(* Logix 5000 project; controller Final vendor 1 type 14 code 242 rev 32.11; software revision 32.00 *)

TASK InitializationTask (periodic, rate 10 ms, priority 10, watchdog 500 ms) : InitializationProgram   // Initializes the tags with default values
TASK MainTask (continuous, watchdog 500 ms) : MainProgram
TASK ProcessDataTask (periodic, rate 10 ms, priority 10, watchdog 500 ms) : ProcessDataI   // Processes the data that has been read and determines the next steps of the pod
TASK ReadTask (periodic, rate 10 ms, priority 10, watchdog 500 ms) : UpdatePrev, UpdateCurrent   // Task that reads current sensor values without erasing previous sensor values
TASK SafetyTask (periodic, rate 20 ms, priority 10, watchdog 20 ms, safety) : SafetyProgram

MODULES
   Local : vendor 1 type 14 code 242 (5069 0, rev 32.11)
      IO_002 : 5069-IF8 (5069 2, rev 2.1, StandardDataDriven RPI 100 ms)
      IO_001 : 5069-IF8 (5069 1, rev 2.1, StandardDataDriven RPI 100 ms)
      IO_003 : 5069-IF8 (5069 3, rev 2.1, StandardDataDriven RPI 100 ms)
      IO_006 : vendor 1 type 7 code 394 (5069 6, rev 2.1, StandardDataDriven RPI 5 ms)
      IO_004 : vendor 1 type 7 code 395 (5069 4, rev 2.1, StandardDataDriven RPI 5 ms)
      IO_005 : vendor 1 type 7 code 395 (5069 5, rev 2.1, StandardDataDriven RPI 5 ms)
      IO_007 : vendor 1 type 109 code 90 (5069 7, rev 3.1, StandardDataDriven RPI 80 ms)
      EN_001 : 1734-AENTR (Ethernet 107.0.114.14, rev 5.1, Output RPI 20 ms)
END_MODULES

TYPE SensorType :   // To monitor the sensor readings, we use this data type
STRUCT
   CurrentValue : DINT;
   PreviousValue0 : DINT;
   PreviousValue1 : DINT;
   PreviousValue2 : DINT;
   PreviousValue3 : DINT;
   PreviousValue4 : DINT;
   PreviousValue5 : DINT;
   PreviousValue6 : DINT;
   PreviousValue7 : DINT;
   PreviousValue8 : DINT;
   PreviousValue9 : DINT;
   Mean10 : DINT;
   StanDev : DINT;
   State : DINT;
   Count : DINT;
END_STRUCT
END_TYPE

VAR_GLOBAL   (* controller tags *)
   B_Pres0 : SensorType;   // Holds all values related to Brakes Pressure Sensor #0
   B_Pres1 : SensorType;   // Holds all values related to Brakes Pressure Sensor #1
   B_Pres2 : SensorType;   // Holds all values related to Brakes Pressure Sensor #2
   B_Pres3 : SensorType;   // Holds all values related to Brakes Pressure Sensor #3
   B_Pres4 : SensorType;   // Holds all values related to Brakes Pressure Sensor #4
   B_Pres5 : SensorType;   // Holds all values related to Brakes Pressure Sensor #5
   B_Pres6 : SensorType;   // Holds all values related to Brakes Pressure Sensor #6
   B_Pres7 : SensorType;   // Holds all values related to Brakes Pressure Sensor #7
   B_Pres8 : SensorType;   // Holds all values related to Brakes Pressure Sensor #8
   B_Pres9 : SensorType;   // Holds all values related to Brakes Pressure Sensor #9
   B_Tem0 : SensorType;   // Holds all values related to Brakes Temperature Sensor #0
   B_Tem1 : SensorType;   // Holds all values related to Brakes Temperature Sensor #1
   C_Las0 : SensorType;   // Holds all values related to Controls Laser Sensor #0
   C_Las1 : SensorType;   // Holds all values related to Controls Laser Sensor #1
   CurrentState : DINT;
   P_Pres0 : SensorType;   // Holds all values related to Pressure Pressure Sensor #0
   P_Pres1 : SensorType;   // Holds all values related to Pressure Pressure Sensor #1
   P_Pres2 : SensorType;   // Holds all values related to Pressure Pressure Sensor #2
   P_Tem0 : SensorType;   // Holds all values related to Pressure Temperature Sensor #0
   P_Tem1 : SensorType;   // Holds all values related to Pressure Temperature Sensor #1
END_VAR

PROGRAM InitializationProgram   (* main routine Initial_B_Pres0 *)

ROUTINE Initial_B_Pres0   (* structured text *)
   B_Pres0.CurrentValue := 0;
   B_Pres0.PreviousValue0 := 0;
   B_Pres0.PreviousValue1 := 0;
   B_Pres0.PreviousValue2 := 0;
   B_Pres0.PreviousValue3 := 0;
   B_Pres0.PreviousValue4 := 0;
   B_Pres0.PreviousValue5 := 0;
   B_Pres0.PreviousValue6 := 0;
   B_Pres0.PreviousValue7 := 0;
   B_Pres0.PreviousValue8 := 0;
   B_Pres0.PreviousValue9 := 0;
   B_Pres0.Count := 0;
   B_Pres0.Mean10 := 0;
   B_Pres0.StanDev := 0;
   B_Pres0.State := 0;
END_ROUTINE

ROUTINE Initial_B_Pres1   (* structured text *)
   B_Pres1.CurrentValue := 0;
   B_Pres1.PreviousValue0 := 0;
   B_Pres1.PreviousValue1 := 0;
   B_Pres1.PreviousValue2 := 0;
   B_Pres1.PreviousValue3 := 0;
   B_Pres1.PreviousValue4 := 0;
   B_Pres1.PreviousValue5 := 0;
   B_Pres1.PreviousValue6 := 0;
   B_Pres1.PreviousValue7 := 0;
   B_Pres1.PreviousValue8 := 0;
   B_Pres1.PreviousValue9 := 0;
   B_Pres1.Count := 0;
   B_Pres1.Mean10 := 0;
   B_Pres1.StanDev := 0;
   B_Pres1.State := 0;
END_ROUTINE

ROUTINE Initial_B_Pres2   (* structured text *)
   B_Pres2.CurrentValue := 0;
   B_Pres2.PreviousValue0 := 0;
   B_Pres2.PreviousValue1 := 0;
   B_Pres2.PreviousValue2 := 0;
   B_Pres2.PreviousValue3 := 0;
   B_Pres2.PreviousValue4 := 0;
   B_Pres2.PreviousValue5 := 0;
   B_Pres2.PreviousValue6 := 0;
   B_Pres2.PreviousValue7 := 0;
   B_Pres2.PreviousValue8 := 0;
   B_Pres2.PreviousValue9 := 0;
   B_Pres2.Count := 0;
   B_Pres2.Mean10 := 0;
   B_Pres2.StanDev := 0;
   B_Pres2.State := 0;
END_ROUTINE

ROUTINE Initial_B_Pres3   (* structured text *)
   B_Pres3.CurrentValue := 0;
   B_Pres3.PreviousValue0 := 0;
   B_Pres3.PreviousValue1 := 0;
   B_Pres3.PreviousValue2 := 0;
   B_Pres3.PreviousValue3 := 0;
   B_Pres3.PreviousValue4 := 0;
   B_Pres3.PreviousValue5 := 0;
   B_Pres3.PreviousValue6 := 0;
   B_Pres3.PreviousValue7 := 0;
   B_Pres3.PreviousValue8 := 0;
   B_Pres3.PreviousValue9 := 0;
   B_Pres3.Count := 0;
   B_Pres3.Mean10 := 0;
   B_Pres3.StanDev := 0;
   B_Pres3.State := 0;
END_ROUTINE

ROUTINE Initial_B_Pres4   (* structured text *)
   B_Pres4.CurrentValue := 0;
   B_Pres4.PreviousValue0 := 0;
   B_Pres4.PreviousValue1 := 0;
   B_Pres4.PreviousValue2 := 0;
   B_Pres4.PreviousValue3 := 0;
   B_Pres4.PreviousValue4 := 0;
   B_Pres4.PreviousValue5 := 0;
   B_Pres4.PreviousValue6 := 0;
   B_Pres4.PreviousValue7 := 0;
   B_Pres4.PreviousValue8 := 0;
   B_Pres4.PreviousValue9 := 0;
   B_Pres4.Count := 0;
   B_Pres4.Mean10 := 0;
   B_Pres4.StanDev := 0;
   B_Pres4.State := 0;
END_ROUTINE

ROUTINE Initial_B_Pres5   (* structured text *)
   B_Pres5.CurrentValue := 0;
   B_Pres5.PreviousValue0 := 0;
   B_Pres5.PreviousValue1 := 0;
   B_Pres5.PreviousValue2 := 0;
   B_Pres5.PreviousValue3 := 0;
   B_Pres5.PreviousValue4 := 0;
   B_Pres5.PreviousValue5 := 0;
   B_Pres5.PreviousValue6 := 0;
   B_Pres5.PreviousValue7 := 0;
   B_Pres5.PreviousValue8 := 0;
   B_Pres5.PreviousValue9 := 0;
   B_Pres5.Count := 0;
   B_Pres5.Mean10 := 0;
   B_Pres5.StanDev := 0;
   B_Pres5.State := 0;
END_ROUTINE

ROUTINE Initial_B_Pres6   (* structured text *)
   B_Pres6.CurrentValue := 0;
   B_Pres6.PreviousValue0 := 0;
   B_Pres6.PreviousValue1 := 0;
   B_Pres6.PreviousValue2 := 0;
   B_Pres6.PreviousValue3 := 0;
   B_Pres6.PreviousValue4 := 0;
   B_Pres6.PreviousValue5 := 0;
   B_Pres6.PreviousValue6 := 0;
   B_Pres6.PreviousValue7 := 0;
   B_Pres6.PreviousValue8 := 0;
   B_Pres6.PreviousValue9 := 0;
   B_Pres6.Count := 0;
   B_Pres6.Mean10 := 0;
   B_Pres6.StanDev := 0;
   B_Pres6.State := 0;
END_ROUTINE

ROUTINE Initial_B_Pres7   (* structured text *)
   B_Pres7.CurrentValue := 0;
   B_Pres7.PreviousValue0 := 0;
   B_Pres7.PreviousValue1 := 0;
   B_Pres7.PreviousValue2 := 0;
   B_Pres7.PreviousValue3 := 0;
   B_Pres7.PreviousValue4 := 0;
   B_Pres7.PreviousValue5 := 0;
   B_Pres7.PreviousValue6 := 0;
   B_Pres7.PreviousValue7 := 0;
   B_Pres7.PreviousValue8 := 0;
   B_Pres7.PreviousValue9 := 0;
   B_Pres7.Count := 0;
   B_Pres7.Mean10 := 0;
   B_Pres7.StanDev := 0;
   B_Pres7.State := 0;
END_ROUTINE

ROUTINE Initial_B_Pres8   (* structured text *)
   B_Pres8.CurrentValue := 0;
   B_Pres8.PreviousValue0 := 0;
   B_Pres8.PreviousValue1 := 0;
   B_Pres8.PreviousValue2 := 0;
   B_Pres8.PreviousValue3 := 0;
   B_Pres8.PreviousValue4 := 0;
   B_Pres8.PreviousValue5 := 0;
   B_Pres8.PreviousValue6 := 0;
   B_Pres8.PreviousValue7 := 0;
   B_Pres8.PreviousValue8 := 0;
   B_Pres8.PreviousValue9 := 0;
   B_Pres8.Count := 0;
   B_Pres8.Mean10 := 0;
   B_Pres8.StanDev := 0;
   B_Pres8.State := 0;
END_ROUTINE

ROUTINE Initial_B_Pres9   (* structured text *)
   B_Pres9.CurrentValue := 0;
   B_Pres9.PreviousValue0 := 0;
   B_Pres9.PreviousValue1 := 0;
   B_Pres9.PreviousValue2 := 0;
   B_Pres9.PreviousValue3 := 0;
   B_Pres9.PreviousValue4 := 0;
   B_Pres9.PreviousValue5 := 0;
   B_Pres9.PreviousValue6 := 0;
   B_Pres9.PreviousValue7 := 0;
   B_Pres9.PreviousValue8 := 0;
   B_Pres9.PreviousValue9 := 0;
   B_Pres9.Count := 0;
   B_Pres9.Mean10 := 0;
   B_Pres9.StanDev := 0;
   B_Pres9.State := 0;
END_ROUTINE

ROUTINE Initial_B_Tem0   (* structured text *)
   B_Tem0.CurrentValue := 0;
   B_Tem0.PreviousValue0 := 0;
   B_Tem0.PreviousValue1 := 0;
   B_Tem0.PreviousValue2 := 0;
   B_Tem0.PreviousValue3 := 0;
   B_Tem0.PreviousValue4 := 0;
   B_Tem0.PreviousValue5 := 0;
   B_Tem0.PreviousValue6 := 0;
   B_Tem0.PreviousValue7 := 0;
   B_Tem0.PreviousValue8 := 0;
   B_Tem0.PreviousValue9 := 0;
   B_Tem0.Count := 0;
   B_Tem0.Mean10 := 0;
   B_Tem0.StanDev := 0;
   B_Tem0.State := 0;
END_ROUTINE

ROUTINE Initial_B_Tem1   (* structured text *)
   B_Tem1.CurrentValue := 0;
   B_Tem1.PreviousValue0 := 0;
   B_Tem1.PreviousValue1 := 0;
   B_Tem1.PreviousValue2 := 0;
   B_Tem1.PreviousValue3 := 0;
   B_Tem1.PreviousValue4 := 0;
   B_Tem1.PreviousValue5 := 0;
   B_Tem1.PreviousValue6 := 0;
   B_Tem1.PreviousValue7 := 0;
   B_Tem1.PreviousValue8 := 0;
   B_Tem1.PreviousValue9 := 0;
   B_Tem1.Count := 0;
   B_Tem1.Mean10 := 0;
   B_Tem1.StanDev := 0;
   B_Tem1.State := 0;
END_ROUTINE

ROUTINE Initial_C_Las0   (* structured text *)
   C_Las0.CurrentValue := 0;
   C_Las0.PreviousValue0 := 0;
   C_Las0.PreviousValue1 := 0;
   C_Las0.PreviousValue2 := 0;
   C_Las0.PreviousValue3 := 0;
   C_Las0.PreviousValue4 := 0;
   C_Las0.PreviousValue5 := 0;
   C_Las0.PreviousValue6 := 0;
   C_Las0.PreviousValue7 := 0;
   C_Las0.PreviousValue8 := 0;
   C_Las0.PreviousValue9 := 0;
   C_Las0.Count := 0;
   C_Las0.Mean10 := 0;
   C_Las0.StanDev := 0;
   C_Las0.State := 0;
END_ROUTINE

ROUTINE Initial_C_Las1   (* structured text *)
   C_Las1.CurrentValue := 0;
   C_Las1.PreviousValue0 := 0;
   C_Las1.PreviousValue1 := 0;
   C_Las1.PreviousValue2 := 0;
   C_Las1.PreviousValue3 := 0;
   C_Las1.PreviousValue4 := 0;
   C_Las1.PreviousValue5 := 0;
   C_Las1.PreviousValue6 := 0;
   C_Las1.PreviousValue7 := 0;
   C_Las1.PreviousValue8 := 0;
   C_Las1.PreviousValue9 := 0;
   C_Las1.Count := 0;
   C_Las1.Mean10 := 0;
   C_Las1.StanDev := 0;
   C_Las1.State := 0;
END_ROUTINE

ROUTINE Initial_P_Pres0   (* structured text *)
   P_Pres0.CurrentValue := 0;
   P_Pres0.PreviousValue0 := 0;
   P_Pres0.PreviousValue1 := 0;
   P_Pres0.PreviousValue2 := 0;
   P_Pres0.PreviousValue3 := 0;
   P_Pres0.PreviousValue4 := 0;
   P_Pres0.PreviousValue5 := 0;
   P_Pres0.PreviousValue6 := 0;
   P_Pres0.PreviousValue7 := 0;
   P_Pres0.PreviousValue8 := 0;
   P_Pres0.PreviousValue9 := 0;
   P_Pres0.Count := 0;
   P_Pres0.Mean10 := 0;
   P_Pres0.StanDev := 0;
   P_Pres0.State := 0;
END_ROUTINE

ROUTINE Initial_P_Pres1   (* structured text *)
   P_Pres1.CurrentValue := 0;
   P_Pres1.PreviousValue0 := 0;
   P_Pres1.PreviousValue1 := 0;
   P_Pres1.PreviousValue2 := 0;
   P_Pres1.PreviousValue3 := 0;
   P_Pres1.PreviousValue4 := 0;
   P_Pres1.PreviousValue5 := 0;
   P_Pres1.PreviousValue6 := 0;
   P_Pres1.PreviousValue7 := 0;
   P_Pres1.PreviousValue8 := 0;
   P_Pres1.PreviousValue9 := 0;
   P_Pres1.Count := 0;
   P_Pres1.Mean10 := 0;
   P_Pres1.StanDev := 0;
   P_Pres1.State := 0;
END_ROUTINE

ROUTINE Initial_P_Pres2   (* structured text *)
   P_Pres2.CurrentValue := 0;
   P_Pres2.PreviousValue0 := 0;
   P_Pres2.PreviousValue1 := 0;
   P_Pres2.PreviousValue2 := 0;
   P_Pres2.PreviousValue3 := 0;
   P_Pres2.PreviousValue4 := 0;
   P_Pres2.PreviousValue5 := 0;
   P_Pres2.PreviousValue6 := 0;
   P_Pres2.PreviousValue7 := 0;
   P_Pres2.PreviousValue8 := 0;
   P_Pres2.PreviousValue9 := 0;
   P_Pres2.Count := 0;
   P_Pres2.Mean10 := 0;
   P_Pres2.StanDev := 0;
   P_Pres2.State := 0;
END_ROUTINE

ROUTINE Initial_P_Tem0   (* structured text *)
   P_Tem0.CurrentValue := 0;
   P_Tem0.PreviousValue0 := 0;
   P_Tem0.PreviousValue1 := 0;
   P_Tem0.PreviousValue2 := 0;
   P_Tem0.PreviousValue3 := 0;
   P_Tem0.PreviousValue4 := 0;
   P_Tem0.PreviousValue5 := 0;
   P_Tem0.PreviousValue6 := 0;
   P_Tem0.PreviousValue7 := 0;
   P_Tem0.PreviousValue8 := 0;
   P_Tem0.PreviousValue9 := 0;
   P_Tem0.Count := 0;
   P_Tem0.Mean10 := 0;
   P_Tem0.StanDev := 0;
   P_Tem0.State := 0;
END_ROUTINE

ROUTINE Initial_P_Tem1   (* structured text *)
   P_Tem1.CurrentValue := 0;
   P_Tem1.PreviousValue0 := 0;
   P_Tem1.PreviousValue1 := 0;
   P_Tem1.PreviousValue2 := 0;
   P_Tem1.PreviousValue3 := 0;
   P_Tem1.PreviousValue4 := 0;
   P_Tem1.PreviousValue5 := 0;
   P_Tem1.PreviousValue6 := 0;
   P_Tem1.PreviousValue7 := 0;
   P_Tem1.PreviousValue8 := 0;
   P_Tem1.PreviousValue9 := 0;
   P_Tem1.Count := 0;
   P_Tem1.Mean10 := 0;
   P_Tem1.StanDev := 0;
   P_Tem1.State := 0;
END_ROUTINE
END_PROGRAM

PROGRAM MainProgram   (* main routine MainRoutine *)

ROUTINE MainRoutine   (* ladder *)
END_ROUTINE
END_PROGRAM

PROGRAM ProcessDataI   (* main routine R001 *)
// Part-I of Process Data
VAR
   acceleration : DINT;
   crawl_distance_brake : DINT;
   distance : DINT;
   distance_brake : DINT;
   getDistance : DINT;
   nominal_count : DINT;
   prev_distance : DINT;
   prev_time : DINT;
   prev_velocity : DINT;
   temp_distance : DINT;
   time : DINT;
   velocity : DINT;
END_VAR

ROUTINE R001   (* structured text *)
   prev_time := time;
   prev_distance := distance;
   prev_velocity := velocity;
   time :=  TT;
   
   temp_distance := 0;
   nominal_count := 0;
   IF C_Las0.State = 0 THEN
               temp_distance :=  C_Las0.CurrentValue;
               nominal_count := 1;
   END_IF;
    IF C_Las1.State = 0 THEN
               temp_distance := temp_distance + C_Las1.CurrentValue;
               nominal_count := nominal_count + 1;
    END_IF;
   temp_distance := temp_distance / nominal_count;
   getDistance := temp_distance;
   
   distance := getDistance;
   velocity := (distance - prev_distance)/(time - prev_time);
   acceleration := (velocity - prev_velocity)/(time - prev_time);
END_ROUTINE

ROUTINE R002   (* structured text *)
   CASE EN_001:I.Data of
               1:  CurrentState := 1;
               2:  CurrentState := 0;
               3:  CurrentState := 2;
               4:  CurrentState := 3;
               6:  CurrentState := 5;
               8:  CurrentState := 6;
               10: CurrentState := 8;
    END_CASE;
END_ROUTINE

ROUTINE R003   (* structured text *)
   IF distance = (distance_brake) THEN
   	CurrentState := 5;
   ELSIF distance = (crawl_distance_brake) THEN
   	CurrentState := 5;
   //elsif timer
   END_IF;
    IF acceleration = 0 THEN
   	CurrentState := 4;
   //elsif timer
   END_IF;
   IF velocity = 0 THEN
   	CurrentState := 7;
   END_IF;
END_ROUTINE
END_PROGRAM

PROGRAM SafetyProgram   (* main routine MainRoutine, safety *)

ROUTINE MainRoutine   (* ladder *)
END_ROUTINE
END_PROGRAM

PROGRAM UpdateCurrent   (* main routine UC_B_Pres0 *)
// Program to store current sensor values
VAR
   range0 : DINT;
   range1 : DINT;
   range2 : DINT;
   range3 : DINT;
   range4 : DINT;
   range5 : DINT;
   range6 : DINT;
   range7 : DINT;
END_VAR

ROUTINE UC_B_Pres0   (* structured text *)
   B_Pres0.CurrentValue := Local:1:I.Ch00.Data;
END_ROUTINE

ROUTINE UC_B_Pres1   (* structured text *)
   B_Pres1.CurrentValue := Local:1:I.Ch01.Data;
END_ROUTINE

ROUTINE UC_B_Pres2   (* structured text *)
   B_Pres2.CurrentValue := Local:1:I.Ch02.Data;
END_ROUTINE

ROUTINE UC_B_Pres3   (* structured text *)
   B_Pres3.CurrentValue := Local:1:I.Ch03.Data;
END_ROUTINE

ROUTINE UC_B_Pres4   (* structured text *)
   B_Pres4.CurrentValue := Local:1:I.Ch04.Data;
END_ROUTINE

ROUTINE UC_B_Pres5   (* structured text *)
   B_Pres5.CurrentValue := Local:1:I.Ch05.Data;
END_ROUTINE

ROUTINE UC_B_Pres6   (* structured text *)
   B_Pres6.CurrentValue := Local:1:I.Ch06.Data;
END_ROUTINE

ROUTINE UC_B_Pres7   (* structured text *)
   B_Pres7.CurrentValue := Local:1:I.Ch07.Data;
END_ROUTINE

ROUTINE UC_B_Pres8   (* structured text *)
   B_Pres8.CurrentValue := Local:2:I.Ch00.Data;
END_ROUTINE

ROUTINE UC_B_Pres9   (* structured text *)
   B_Pres9.CurrentValue := Local:2:I.Ch01.Data;
END_ROUTINE

ROUTINE UC_B_Tem0   (* structured text *)
   B_Tem0.CurrentValue := Local:2:I.Ch02.Data;
END_ROUTINE

ROUTINE UC_B_Tem1   (* structured text *)
   B_Tem1.CurrentValue := Local:2:I.Ch03.Data;
END_ROUTINE

ROUTINE UC_C_Las0   (* structured text *)
   C_Las0.CurrentValue := Local:7:I.Output00;
END_ROUTINE

ROUTINE UC_C_Las1   (* structured text *)
   C_Las1.CurrentValue := Local:7:I.Output01;
END_ROUTINE

ROUTINE UC_P_Pres0   (* structured text *)
   P_Pres0.CurrentValue := Local:3:I.Ch00.Data;
END_ROUTINE

ROUTINE UC_P_Pres1   (* structured text *)
   P_Pres1.CurrentValue := Local:3:I.Ch01.Data;
END_ROUTINE

ROUTINE UC_P_Pres2   (* structured text *)
   P_Pres2.CurrentValue := Local:3:I.Ch02.Data;
END_ROUTINE

ROUTINE UC_P_Tem0   (* structured text *)
   P_Tem0.CurrentValue := Local:3:I.Ch04.Data;
END_ROUTINE

ROUTINE UC_P_Tem1   (* structured text *)
   P_Tem1.CurrentValue := Local:3:I.Ch05.Data;
END_ROUTINE
END_PROGRAM

PROGRAM UpdatePrev   (* main routine UP_B_Pres0 *)
// Program to store previous sensor values

ROUTINE UP_B_Pres0   (* structured text *)
// Routine for Brakes Pressure Sensor #0
   case B_Pres0.Count of
   	0: B_Pres0.PreviousValue0 := B_Pres0.CurrentValue;
   	1: B_Pres0.PreviousValue1 := B_Pres0.CurrentValue;
   	2: B_Pres0.PreviousValue2 := B_Pres0.CurrentValue;
   	3: B_Pres0.PreviousValue3 := B_Pres0.CurrentValue;
   	4: B_Pres0.PreviousValue4 := B_Pres0.CurrentValue;
   	5: B_Pres0.PreviousValue5 := B_Pres0.CurrentValue;
   	6: B_Pres0.PreviousValue6 := B_Pres0.CurrentValue;
   	7: B_Pres0.PreviousValue7 := B_Pres0.CurrentValue;
   	8: B_Pres0.PreviousValue8 := B_Pres0.CurrentValue;
   	9: B_Pres0.PreviousValue9 := B_Pres0.CurrentValue;
   end_case;
   B_Pres0.Count = B_Pres0.Count + 1;
   if B_Pres0.Count = 10 then
   	B_Pres0.Count = 0;
   end_if;
END_ROUTINE

ROUTINE UP_B_Pres1   (* structured text *)
   case B_Pres1.Count of
   	0: B_Pres1.PreviousValue0 := B_Pres1.CurrentValue;
   	1: B_Pres1.PreviousValue1 := B_Pres1.CurrentValue;
   	2: B_Pres1.PreviousValue2 := B_Pres1.CurrentValue;
   	3: B_Pres1.PreviousValue3 := B_Pres1.CurrentValue;
   	4: B_Pres1.PreviousValue4 := B_Pres1.CurrentValue;
   	5: B_Pres1.PreviousValue5 := B_Pres1.CurrentValue;
   	6: B_Pres1.PreviousValue6 := B_Pres1.CurrentValue;
   	7: B_Pres1.PreviousValue7 := B_Pres1.CurrentValue;
   	8: B_Pres1.PreviousValue8 := B_Pres1.CurrentValue;
   	9: B_Pres1.PreviousValue9 := B_Pres1.CurrentValue;
   end_case;
   B_Pres1.Count = B_Pres1.Count + 1;
   if B_Pres1.Count = 10 then
   	B_Pres1.Count = 0;
   end_if;
END_ROUTINE

ROUTINE UP_B_Pres2   (* structured text *)
   case B_Pres2.Count of
   	0: B_Pres2.PreviousValue0 := B_Pres2.CurrentValue;
   	1: B_Pres2.PreviousValue1 := B_Pres2.CurrentValue;
   	2: B_Pres2.PreviousValue2 := B_Pres2.CurrentValue;
   	3: B_Pres2.PreviousValue3 := B_Pres2.CurrentValue;
   	4: B_Pres2.PreviousValue4 := B_Pres2.CurrentValue;
   	5: B_Pres2.PreviousValue5 := B_Pres2.CurrentValue;
   	6: B_Pres2.PreviousValue6 := B_Pres2.CurrentValue;
   	7: B_Pres2.PreviousValue7 := B_Pres2.CurrentValue;
   	8: B_Pres2.PreviousValue8 := B_Pres2.CurrentValue;
   	9: B_Pres2.PreviousValue9 := B_Pres2.CurrentValue;
   end_case;
   B_Pres2.Count = B_Pres2.Count + 1;
   if B_Pres2.Count = 10 then
   	B_Pres2.Count = 0;
   end_if;
END_ROUTINE

ROUTINE UP_B_Pres3   (* structured text *)
   case B_Pres3.Count of
   	0: B_Pres3.PreviousValue0 := B_Pres3.CurrentValue;
   	1: B_Pres3.PreviousValue1 := B_Pres3.CurrentValue;
   	2: B_Pres3.PreviousValue2 := B_Pres3.CurrentValue;
   	3: B_Pres3.PreviousValue3 := B_Pres3.CurrentValue;
   	4: B_Pres3.PreviousValue4 := B_Pres3.CurrentValue;
   	5: B_Pres3.PreviousValue5 := B_Pres3.CurrentValue;
   	6: B_Pres3.PreviousValue6 := B_Pres3.CurrentValue;
   	7: B_Pres3.PreviousValue7 := B_Pres3.CurrentValue;
   	8: B_Pres3.PreviousValue8 := B_Pres3.CurrentValue;
   	9: B_Pres3.PreviousValue9 := B_Pres3.CurrentValue;
   end_case;
   B_Pres3.Count = B_Pres3.Count + 1;
   if B_Pres3.Count = 10 then
   	B_Pres3.Count = 0;
   end_if;
END_ROUTINE

ROUTINE UP_B_Pres4   (* structured text *)
   case B_Pres4.Count of
   	0: B_Pres4.PreviousValue0 := B_Pres4.CurrentValue;
   	1: B_Pres4.PreviousValue1 := B_Pres4.CurrentValue;
   	2: B_Pres4.PreviousValue2 := B_Pres4.CurrentValue;
   	3: B_Pres4.PreviousValue3 := B_Pres4.CurrentValue;
   	4: B_Pres4.PreviousValue4 := B_Pres4.CurrentValue;
   	5: B_Pres4.PreviousValue5 := B_Pres4.CurrentValue;
   	6: B_Pres4.PreviousValue6 := B_Pres4.CurrentValue;
   	7: B_Pres4.PreviousValue7 := B_Pres4.CurrentValue;
   	8: B_Pres4.PreviousValue8 := B_Pres4.CurrentValue;
   	9: B_Pres4.PreviousValue9 := B_Pres4.CurrentValue;
   end_case;
   B_Pres4.Count = B_Pres4.Count + 1;
   if B_Pres4.Count = 10 then
   	B_Pres4.Count = 0;
   end_if;
END_ROUTINE

ROUTINE UP_B_Pres5   (* structured text *)
   case B_Pres5.Count of
   	0: B_Pres5.PreviousValue0 := B_Pres5.CurrentValue;
   	1: B_Pres5.PreviousValue1 := B_Pres5.CurrentValue;
   	2: B_Pres5.PreviousValue2 := B_Pres5.CurrentValue;
   	3: B_Pres5.PreviousValue3 := B_Pres5.CurrentValue;
   	4: B_Pres5.PreviousValue4 := B_Pres5.CurrentValue;
   	5: B_Pres5.PreviousValue5 := B_Pres5.CurrentValue;
   	6: B_Pres5.PreviousValue6 := B_Pres5.CurrentValue;
   	7: B_Pres5.PreviousValue7 := B_Pres5.CurrentValue;
   	8: B_Pres5.PreviousValue8 := B_Pres5.CurrentValue;
   	9: B_Pres5.PreviousValue9 := B_Pres5.CurrentValue;
   end_case;
   B_Pres5.Count = B_Pres5.Count + 1;
   if B_Pres5.Count = 10 then
   	B_Pres5.Count = 0;
   end_if;
END_ROUTINE

ROUTINE UP_B_Pres6   (* structured text *)
   case B_Pres6.Count of
   	0: B_Pres6.PreviousValue0 := B_Pres6.CurrentValue;
   	1: B_Pres6.PreviousValue1 := B_Pres6.CurrentValue;
   	2: B_Pres6.PreviousValue2 := B_Pres6.CurrentValue;
   	3: B_Pres6.PreviousValue3 := B_Pres6.CurrentValue;
   	4: B_Pres6.PreviousValue4 := B_Pres6.CurrentValue;
   	5: B_Pres6.PreviousValue5 := B_Pres6.CurrentValue;
   	6: B_Pres6.PreviousValue6 := B_Pres6.CurrentValue;
   	7: B_Pres6.PreviousValue7 := B_Pres6.CurrentValue;
   	8: B_Pres6.PreviousValue8 := B_Pres6.CurrentValue;
   	9: B_Pres6.PreviousValue9 := B_Pres6.CurrentValue;
   end_case;
   B_Pres6.Count = B_Pres6.Count + 1;
   if B_Pres6.Count = 10 then
   	B_Pres6.Count = 0;
   end_if;
END_ROUTINE

ROUTINE UP_B_Pres7   (* structured text *)
   case B_Pres7.Count of
   	0: B_Pres7.PreviousValue0 := B_Pres7.CurrentValue;
   	1: B_Pres7.PreviousValue1 := B_Pres7.CurrentValue;
   	2: B_Pres7.PreviousValue2 := B_Pres7.CurrentValue;
   	3: B_Pres7.PreviousValue3 := B_Pres7.CurrentValue;
   	4: B_Pres7.PreviousValue4 := B_Pres7.CurrentValue;
   	5: B_Pres7.PreviousValue5 := B_Pres7.CurrentValue;
   	6: B_Pres7.PreviousValue6 := B_Pres7.CurrentValue;
   	7: B_Pres7.PreviousValue7 := B_Pres7.CurrentValue;
   	8: B_Pres7.PreviousValue8 := B_Pres7.CurrentValue;
   	9: B_Pres7.PreviousValue9 := B_Pres7.CurrentValue;
   end_case;
   B_Pres7.Count = B_Pres7.Count + 1;
   if B_Pres7.Count = 10 then
   	B_Pres7.Count = 0;
   end_if;
END_ROUTINE

ROUTINE UP_B_Pres8   (* structured text *)
   case B_Pres8.Count of
   	0: B_Pres8.PreviousValue0 := B_Pres8.CurrentValue;
   	1: B_Pres8.PreviousValue1 := B_Pres8.CurrentValue;
   	2: B_Pres8.PreviousValue2 := B_Pres8.CurrentValue;
   	3: B_Pres8.PreviousValue3 := B_Pres8.CurrentValue;
   	4: B_Pres8.PreviousValue4 := B_Pres8.CurrentValue;
   	5: B_Pres8.PreviousValue5 := B_Pres8.CurrentValue;
   	6: B_Pres8.PreviousValue6 := B_Pres8.CurrentValue;
   	7: B_Pres8.PreviousValue7 := B_Pres8.CurrentValue;
   	8: B_Pres8.PreviousValue8 := B_Pres8.CurrentValue;
   	9: B_Pres8.PreviousValue9 := B_Pres8.CurrentValue;
   end_case;
   B_Pres8.Count = B_Pres8.Count + 1;
   if B_Pres8.Count = 10 then
   	B_Pres8.Count = 0;
   end_if;
END_ROUTINE

ROUTINE UP_B_Pres9   (* structured text *)
   case B_Pres9.Count of
   	0: B_Pres9.PreviousValue0 := B_Pres9.CurrentValue;
   	1: B_Pres9.PreviousValue1 := B_Pres9.CurrentValue;
   	2: B_Pres9.PreviousValue2 := B_Pres9.CurrentValue;
   	3: B_Pres9.PreviousValue3 := B_Pres9.CurrentValue;
   	4: B_Pres9.PreviousValue4 := B_Pres9.CurrentValue;
   	5: B_Pres9.PreviousValue5 := B_Pres9.CurrentValue;
   	6: B_Pres9.PreviousValue6 := B_Pres9.CurrentValue;
   	7: B_Pres9.PreviousValue7 := B_Pres9.CurrentValue;
   	8: B_Pres9.PreviousValue8 := B_Pres9.CurrentValue;
   	9: B_Pres9.PreviousValue9 := B_Pres9.CurrentValue;
   end_case;
   B_Pres9.Count = B_Pres9.Count + 1;
   if B_Pres9.Count = 10 then
   	B_Pres9.Count = 0;
   end_if;
END_ROUTINE

ROUTINE UP_B_Tem0   (* structured text *)
   case B_Tem0.Count of
   	0: B_Tem0.PreviousValue0 := B_Tem0.CurrentValue;
   	1: B_Tem0.PreviousValue1 := B_Tem0.CurrentValue;
   	2: B_Tem0.PreviousValue2 := B_Tem0.CurrentValue;
   	3: B_Tem0.PreviousValue3 := B_Tem0.CurrentValue;
   	4: B_Tem0.PreviousValue4 := B_Tem0.CurrentValue;
   	5: B_Tem0.PreviousValue5 := B_Tem0.CurrentValue;
   	6: B_Tem0.PreviousValue6 := B_Tem0.CurrentValue;
   	7: B_Tem0.PreviousValue7 := B_Tem0.CurrentValue;
   	8: B_Tem0.PreviousValue8 := B_Tem0.CurrentValue;
   	9: B_Tem0.PreviousValue9 := B_Tem0.CurrentValue;
   end_case;
   B_Tem0.Count = B_Tem0.Count + 1;
   if B_Tem0.Count = 10 then
   	B_Tem0.Count = 0;
   end_if;
END_ROUTINE

ROUTINE UP_B_Tem1   (* structured text *)
   case B_Tem1.Count of
   	0: B_Tem1.PreviousValue0 := B_Tem1.CurrentValue;
   	1: B_Tem1.PreviousValue1 := B_Tem1.CurrentValue;
   	2: B_Tem1.PreviousValue2 := B_Tem1.CurrentValue;
   	3: B_Tem1.PreviousValue3 := B_Tem1.CurrentValue;
   	4: B_Tem1.PreviousValue4 := B_Tem1.CurrentValue;
   	5: B_Tem1.PreviousValue5 := B_Tem1.CurrentValue;
   	6: B_Tem1.PreviousValue6 := B_Tem1.CurrentValue;
   	7: B_Tem1.PreviousValue7 := B_Tem1.CurrentValue;
   	8: B_Tem1.PreviousValue8 := B_Tem1.CurrentValue;
   	9: B_Tem1.PreviousValue9 := B_Tem1.CurrentValue;
   end_case;
   B_Tem1.Count = B_Tem1.Count + 1;
   if B_Tem1.Count = 10 then
   	B_Tem1.Count = 0;
   end_if;
END_ROUTINE

ROUTINE UP_C_Las0   (* structured text *)
   case C_Las0.Count of
   	0: C_Las0.PreviousValue0 := C_Las0.CurrentValue;
   	1: C_Las0.PreviousValue1 := C_Las0.CurrentValue;
   	2: C_Las0.PreviousValue2 := C_Las0.CurrentValue;
   	3: C_Las0.PreviousValue3 := C_Las0.CurrentValue;
   	4: C_Las0.PreviousValue4 := C_Las0.CurrentValue;
   	5: C_Las0.PreviousValue5 := C_Las0.CurrentValue;
   	6: C_Las0.PreviousValue6 := C_Las0.CurrentValue;
   	7: C_Las0.PreviousValue7 := C_Las0.CurrentValue;
   	8: C_Las0.PreviousValue8 := C_Las0.CurrentValue;
   	9: C_Las0.PreviousValue9 := C_Las0.CurrentValue;
   end_case;
   C_Las0.Count = C_Las0.Count + 1;
   if C_Las0.Count = 10 then
   	C_Las0.Count = 0;
   end_if;
END_ROUTINE

ROUTINE UP_C_Las1   (* structured text *)
   case C_Las1.Count of
   	0: C_Las1.PreviousValue0 := C_Las1.CurrentValue;
   	1: C_Las1.PreviousValue1 := C_Las1.CurrentValue;
   	2: C_Las1.PreviousValue2 := C_Las1.CurrentValue;
   	3: C_Las1.PreviousValue3 := C_Las1.CurrentValue;
   	4: C_Las1.PreviousValue4 := C_Las1.CurrentValue;
   	5: C_Las1.PreviousValue5 := C_Las1.CurrentValue;
   	6: C_Las1.PreviousValue6 := C_Las1.CurrentValue;
   	7: C_Las1.PreviousValue7 := C_Las1.CurrentValue;
   	8: C_Las1.PreviousValue8 := C_Las1.CurrentValue;
   	9: C_Las1.PreviousValue9 := C_Las1.CurrentValue;
   end_case;
   C_Las1.Count = C_Las1.Count + 1;
   if C_Las1.Count = 10 then
   	C_Las1.Count = 0;
   end_if;
END_ROUTINE

ROUTINE UP_P_Pres0   (* structured text *)
   case P_Pres0.Count of
   	0: P_Pres0.PreviousValue0 := P_Pres0.CurrentValue;
   	1: P_Pres0.PreviousValue1 := P_Pres0.CurrentValue;
   	2: P_Pres0.PreviousValue2 := P_Pres0.CurrentValue;
   	3: P_Pres0.PreviousValue3 := P_Pres0.CurrentValue;
   	4: P_Pres0.PreviousValue4 := P_Pres0.CurrentValue;
   	5: P_Pres0.PreviousValue5 := P_Pres0.CurrentValue;
   	6: P_Pres0.PreviousValue6 := P_Pres0.CurrentValue;
   	7: P_Pres0.PreviousValue7 := P_Pres0.CurrentValue;
   	8: P_Pres0.PreviousValue8 := P_Pres0.CurrentValue;
   	9: P_Pres0.PreviousValue9 := P_Pres0.CurrentValue;
   end_case;
   P_Pres0.Count = P_Pres0.Count + 1;
   if P_Pres0.Count = 10 then
   	P_Pres0.Count = 0;
   end_if;
END_ROUTINE

ROUTINE UP_P_Pres1   (* structured text *)
   case P_Pres1.Count of
   	0: P_Pres1.PreviousValue0 := P_Pres1.CurrentValue;
   	1: P_Pres1.PreviousValue1 := P_Pres1.CurrentValue;
   	2: P_Pres1.PreviousValue2 := P_Pres1.CurrentValue;
   	3: P_Pres1.PreviousValue3 := P_Pres1.CurrentValue;
   	4: P_Pres1.PreviousValue4 := P_Pres1.CurrentValue;
   	5: P_Pres1.PreviousValue5 := P_Pres1.CurrentValue;
   	6: P_Pres1.PreviousValue6 := P_Pres1.CurrentValue;
   	7: P_Pres1.PreviousValue7 := P_Pres1.CurrentValue;
   	8: P_Pres1.PreviousValue8 := P_Pres1.CurrentValue;
   	9: P_Pres1.PreviousValue9 := P_Pres1.CurrentValue;
   end_case;
   P_Pres1.Count = P_Pres1.Count + 1;
   if P_Pres1.Count = 10 then
   	P_Pres1.Count = 0;
   end_if;
END_ROUTINE

ROUTINE UP_P_Pres2   (* structured text *)
   case P_Pres2.Count of
   	0: P_Pres2.PreviousValue0 := P_Pres2.CurrentValue;
   	1: P_Pres2.PreviousValue1 := P_Pres2.CurrentValue;
   	2: P_Pres2.PreviousValue2 := P_Pres2.CurrentValue;
   	3: P_Pres2.PreviousValue3 := P_Pres2.CurrentValue;
   	4: P_Pres2.PreviousValue4 := P_Pres2.CurrentValue;
   	5: P_Pres2.PreviousValue5 := P_Pres2.CurrentValue;
   	6: P_Pres2.PreviousValue6 := P_Pres2.CurrentValue;
   	7: P_Pres2.PreviousValue7 := P_Pres2.CurrentValue;
   	8: P_Pres2.PreviousValue8 := P_Pres2.CurrentValue;
   	9: P_Pres2.PreviousValue9 := P_Pres2.CurrentValue;
   end_case;
   P_Pres2.Count = P_Pres2.Count + 1;
   if P_Pres2.Count = 10 then
   	P_Pres2.Count = 0;
   end_if;
END_ROUTINE

ROUTINE UP_P_Tem0   (* structured text *)
   case P_Tem0.Count of
   	0: P_Tem0.PreviousValue0 := P_Tem0.CurrentValue;
   	1: P_Tem0.PreviousValue1 := P_Tem0.CurrentValue;
   	2: P_Tem0.PreviousValue2 := P_Tem0.CurrentValue;
   	3: P_Tem0.PreviousValue3 := P_Tem0.CurrentValue;
   	4: P_Tem0.PreviousValue4 := P_Tem0.CurrentValue;
   	5: P_Tem0.PreviousValue5 := P_Tem0.CurrentValue;
   	6: P_Tem0.PreviousValue6 := P_Tem0.CurrentValue;
   	7: P_Tem0.PreviousValue7 := P_Tem0.CurrentValue;
   	8: P_Tem0.PreviousValue8 := P_Tem0.CurrentValue;
   	9: P_Tem0.PreviousValue9 := P_Tem0.CurrentValue;
   end_case;
   P_Tem0.Count = P_Tem0.Count + 1;
   if P_Tem0.Count = 10 then
   	P_Tem0.Count = 0;
   end_if;
END_ROUTINE

ROUTINE UP_P_Tem1   (* structured text *)
   case P_Tem1.Count of
   	0: P_Tem1.PreviousValue0 := P_Tem1.CurrentValue;
   	1: P_Tem1.PreviousValue1 := P_Tem1.CurrentValue;
   	2: P_Tem1.PreviousValue2 := P_Tem1.CurrentValue;
   	3: P_Tem1.PreviousValue3 := P_Tem1.CurrentValue;
   	4: P_Tem1.PreviousValue4 := P_Tem1.CurrentValue;
   	5: P_Tem1.PreviousValue5 := P_Tem1.CurrentValue;
   	6: P_Tem1.PreviousValue6 := P_Tem1.CurrentValue;
   	7: P_Tem1.PreviousValue7 := P_Tem1.CurrentValue;
   	8: P_Tem1.PreviousValue8 := P_Tem1.CurrentValue;
   	9: P_Tem1.PreviousValue9 := P_Tem1.CurrentValue;
   end_case;
   P_Tem1.Count = P_Tem1.Count + 1;
   if P_Tem1.Count = 10 then
   	P_Tem1.Count = 0;
   end_if;
END_ROUTINE
END_PROGRAM
